(* IEC 61131-3 sources: CodesysTest/alpha/export/FBs/Components/Motors/Applied Motion/FB_AppliedMotionBagDeliveryMotor_1.pou, 13 files *)

(* ---- FB_AppliedMotionBagDeliveryMotor_1.pou.st ---- *)
(*#-#-#-#-#-#-#-#-#-#---Declaration---#-#-#-#-#-#-#-#-#-#-#-#-#*)

FUNCTION_BLOCK FB_AppliedMotionBagDeliveryMotor_1 EXTENDS FB_AppliedMotionStepServoEIPBase
VAR_INPUT
	ack : BOOL;
	placement : BAG_DELIVERY_MOTOR_PLACEMENT;
	intercommunications : BAG_DELIVERY_MOTOR_INTERCOMMUNICATION;
END_VAR
VAR_OUTPUT
	ackRequest : BOOL;
	tensionFault : BOOL;
END_VAR
VAR
	_moveDistance : BOOL;
	_moveFinal : BOOL;
	_moveDone : BOOL;
	_delayTimer : TON := (PT := T#10MS);
	_moveDistanceState : AMP_EIP_MOVE_INITIAL_STATES;
	_moveDistanceFinalState : AMP_EIP_MOVE_INITIAL_STATES;
	_tensionFaultDwellTimer : TON;
END_VAR
(*#-#-#-#-#-#-#-#-#-#---Implementation---#-#-#-#-#-#-#-#-#-#-#-#-#*)

(* ---- Execute.m.st ---- *)
(*#-#-#-#-#-#-#-#-#-#---Declaration---#-#-#-#-#-#-#-#-#-#-#-#-#*)

METHOD Execute
VAR_INPUT
END_VAR

(*#-#-#-#-#-#-#-#-#-#---Implementation---#-#-#-#-#-#-#-#-#-#-#-#-#*)

//
SUPER^.Execute();

// Used in state engine to delay between moves
_delayTimer();

// If motor velocity is greater then threshold for 2 seconds, fault
_tensionFaultDwellTimer(IN := ABS(velocity) > VELOCITY_THRESHOLD_FOR_TENSION_FAULT);
IF _tensionFaultDwellTimer.Q AND NOT HMIData.enableDryCycle THEN
	tensionFault := TRUE;
END_IF

// Clear Params
IF _restoreToDefault THEN
	_restoreToDefault := FALSE;
	_state := BAG_DELIVERY_MOVE_STATES.Idle;
	commandSuccessful := FALSE;
	tensionFault := FALSE;
	ackRequest := FALSE;
	ack := FALSE;
END_IF

//
CASE _state OF
	BAG_DELIVERY_MOVE_STATES.Idle:
		IF _moveDistance THEN
			_moveDistance := FALSE;
			_state := BAG_DELIVERY_MOVE_STATES.SetToPointToPointMode;
			commandSuccessful := FALSE;
		END_IF

	BAG_DELIVERY_MOVE_STATES.SetToPointToPointMode:
		IF EIP THEN
			IF RearMotor THEN
				TriggerPointToPointMode();
			END_IF
			IF commandSuccessful OR NOT RearMotor THEN
				commandSuccessful := FALSE;
				_state := BAG_DELIVERY_MOVE_STATES.AckPointToPointMode;
			END_IF
		ELSIF NOT EIP THEN
			sclCommand := SCL_SO;
			parameter1 := O2_H;
			commands.SendHostCommand := TRUE;
			IF commandSuccessful THEN
				commandSuccessful := FALSE;
				_state := BAG_DELIVERY_MOVE_STATES.WaitAfterMovingMotor;
			END_IF
		END_IF

	BAG_DELIVERY_MOVE_STATES.WaitAfterSettingOutputOff:
		IF commandSuccessful THEN
			_state := BAG_DELIVERY_MOVE_STATES.MoveMotor;
		END_IF

	BAG_DELIVERY_MOVE_STATES.AckPointToPointMode:
		_delayTimer.PT := T#10MS;
		_delayTimer.IN := TRUE;
		IF _delayTimer.Q THEN
			ackRequest := TRUE; // Request acknowledgment from parent class
			IF ack THEN // Parent class acknowledges this motor and sibling are ready to move
				ackRequest := FALSE;
				_delayTimer.IN := FALSE;
				_state := BAG_DELIVERY_MOVE_STATES.MoveMotor;
			END_IF
		END_IF

	BAG_DELIVERY_MOVE_STATES.MoveMotor:
		FeedToLength();
		_state := BAG_DELIVERY_MOVE_STATES.WaitAfterMovingMotor;

	BAG_DELIVERY_MOVE_STATES.WaitAfterMovingMotor:
		IF NOT _moveFinal THEN
			IF commandSuccessful THEN
				commandSuccessful := FALSE;
				_moveDone := TRUE;
				_state := BAG_DELIVERY_MOVE_STATES.Idle;
			END_IF
		ELSE
			IF commandSuccessful AND InPosition THEN
				_delayTimer.PT := T#10MS;
				_delayTimer.IN := TRUE;
				IF _delayTimer.Q THEN
					_delayTimer.IN := FALSE;
					commandSuccessful := FALSE;
					_state := BAG_DELIVERY_MOVE_STATES.SetToTorqueMode;
				END_IF
			END_IF
		END_IF

	BAG_DELIVERY_MOVE_STATES.SetToTorqueMode:
		IF EIP THEN
			IF RearMotor THEN
				TriggerTorqueMode();
			END_IF
			IF commandSuccessful OR NOT RearMotor THEN
				commandSuccessful := FALSE;
				_state := BAG_DELIVERY_MOVE_STATES.WaitAfterSettingOutputOn;
			END_IF
		ELSE
			TriggerTorqueMode();
			_state := BAG_DELIVERY_MOVE_STATES.WaitAfterSettingOutputOn;
		END_IF

	BAG_DELIVERY_MOVE_STATES.WaitAfterSettingOutputOn:
		IF EIP THEN
			_delayTimer.PT := T#10MS;
			_delayTimer.IN := TRUE;
			IF _delayTimer.Q THEN
				_moveDone := TRUE;
				_moveFinal := FALSE;
				_delayTimer.IN := FALSE;
				_state := BAG_DELIVERY_MOVE_STATES.Idle;
			END_IF
		ELSE
			IF commandSuccessful THEN
				_moveDone := TRUE;
				_state := BAG_DELIVERY_MOVE_STATES.Idle;
				commandSuccessful := FALSE;
			END_IF
		END_IF
END_CASE

(* ---- FeedToLength.m.st ---- *)
(*#-#-#-#-#-#-#-#-#-#---Declaration---#-#-#-#-#-#-#-#-#-#-#-#-#*)

METHOD FeedToLength
VAR_INPUT
END_VAR
(*#-#-#-#-#-#-#-#-#-#---Implementation---#-#-#-#-#-#-#-#-#-#-#-#-#*)

//
sclCommand := 16#0;
parameter1 := 16#0;
commandSuccessful := FALSE;
commands.FeedToLength := TRUE;

(* ---- Initialize.m.st ---- *)
(*#-#-#-#-#-#-#-#-#-#---Declaration---#-#-#-#-#-#-#-#-#-#-#-#-#*)

METHOD Initialize
VAR_INPUT
END_VAR
(*#-#-#-#-#-#-#-#-#-#---Implementation---#-#-#-#-#-#-#-#-#-#-#-#-#*)

//
_initialize := TRUE;

(* ---- MoveDistance.m.st ---- *)
(*#-#-#-#-#-#-#-#-#-#---Declaration---#-#-#-#-#-#-#-#-#-#-#-#-#*)

METHOD MoveDistance
VAR_INPUT
    distance : REAL;    // Distance to move in inches
    acceleration : INT; // Acceleration in RPM/sec
    deceleration : INT; // Deceleration in RPM/sec
    velocity : INT;     // Velocity in .25RPM
END_VAR(*#-#-#-#-#-#-#-#-#-#---Implementation---#-#-#-#-#-#-#-#-#-#-#-#-#*)

//
IF _initialize OR placement = BAG_DELIVERY_MOTOR_PLACEMENT.Rear AND interconnect = BAG_DELIVERY_IC.CBL THEN
	RETURN;
END_IF

//
_moveDone := FALSE;
_moveDistance := TRUE;
_state := BAG_DELIVERY_MOVE_STATES.Idle;

//
distanceToMoveInSteps := REAL_TO_DINT((distance) * stepsPerInchSetpoint);
IF reversePolarity THEN
    distanceToMoveInSteps := distanceToMoveInSteps * -1;
END_IF

//
commandSuccessful := FALSE;
pointToPointAccelSetpoint := acceleration;
pointToPointDecelSetpoint := deceleration;
currentLimit := defaultCurrentSetpoint;
velocitySetpoint := velocity;

(* ---- MoveDistanceFinal.m.st ---- *)
(*#-#-#-#-#-#-#-#-#-#---Declaration---#-#-#-#-#-#-#-#-#-#-#-#-#*)

METHOD MoveDistanceFinal
VAR_INPUT
    distance : REAL;        //Distance to move in inches
    acceleration : INT;        //Acceleration in RPM/sec
    deceleration : INT;        //Deceleration in RPM/sec
    velocity : INT;            //Velocity in .25RPM
END_VAR

VAR
	_movefin: BOOL;
END_VAR(*#-#-#-#-#-#-#-#-#-#---Implementation---#-#-#-#-#-#-#-#-#-#-#-#-#*)

//
_moveDone := FALSE;
_moveFinal := TRUE;
_stateFinal := BAG_DELIVERY_MOVE_STATES.Idle;

//
distanceToMoveInSteps := REAL_TO_DINT((distance) * stepsPerInchSetpoint);
IF reversePolarity THEN
    distanceToMoveInSteps := distanceToMoveInSteps * -1;
END_IF

//
commandSuccessful := FALSE;
pointToPointAccelSetpoint := acceleration;
pointToPointDecelSetpoint := deceleration;
currentLimit := defaultCurrentSetpoint;
velocitySetpoint := velocity;

(* ---- PrepareForCommand.m.st ---- *)
(*#-#-#-#-#-#-#-#-#-#---Declaration---#-#-#-#-#-#-#-#-#-#-#-#-#*)

METHOD PrepareForCommand
VAR_INPUT
END_VAR
(*#-#-#-#-#-#-#-#-#-#---Implementation---#-#-#-#-#-#-#-#-#-#-#-#-#*)

commandSuccessful := FALSE;

(* ---- SetRearMotorToPoint2Point.m.st ---- *)
(*#-#-#-#-#-#-#-#-#-#---Declaration---#-#-#-#-#-#-#-#-#-#-#-#-#*)

METHOD SetRearMotorToPoint2Point
VAR_INPUT
END_VAR
(*#-#-#-#-#-#-#-#-#-#---Implementation---#-#-#-#-#-#-#-#-#-#-#-#-#*)

commandSuccessful := FALSE;
ExecuteStoredProgram(2);

(* ---- SetRearMotorTorqueValue.m.st ---- *)
(*#-#-#-#-#-#-#-#-#-#---Declaration---#-#-#-#-#-#-#-#-#-#-#-#-#*)

METHOD SetRearMotorTorqueValue
VAR_INPUT
	torque : DINT;
END_VAR
(*#-#-#-#-#-#-#-#-#-#---Implementation---#-#-#-#-#-#-#-#-#-#-#-#-#*)

sclCommand := 16#4743; // GC (Current Command)
parameter1 := torque;

commandSuccessful := FALSE;
commands.SendHostCommand := TRUE;

(* ---- SetRearMotorToTorqueMode.m.st ---- *)
(*#-#-#-#-#-#-#-#-#-#---Declaration---#-#-#-#-#-#-#-#-#-#-#-#-#*)

METHOD SetRearMotorToTorqueMode
VAR_INPUT
END_VAR
(*#-#-#-#-#-#-#-#-#-#---Implementation---#-#-#-#-#-#-#-#-#-#-#-#-#*)

commandSuccessful := FALSE;
ExecuteStoredProgram(3);

(* ---- SetTorqueValue.m.st ---- *)
(*#-#-#-#-#-#-#-#-#-#---Declaration---#-#-#-#-#-#-#-#-#-#-#-#-#*)

METHOD SetTorqueValue
VAR_INPUT
	torque : DINT;
END_VAR
(*#-#-#-#-#-#-#-#-#-#---Implementation---#-#-#-#-#-#-#-#-#-#-#-#-#*)

sclCommand := 16#4743; // GC (Current Command)
parameter1 := torque;

commandSuccessful := FALSE;
commands.SendHostCommand := TRUE;

(* ---- TriggerPointToPointMode.m.st ---- *)
(*#-#-#-#-#-#-#-#-#-#---Declaration---#-#-#-#-#-#-#-#-#-#-#-#-#*)

METHOD TriggerPointToPointMode
VAR_INPUT
END_VAR

(*#-#-#-#-#-#-#-#-#-#---Implementation---#-#-#-#-#-#-#-#-#-#-#-#-#*)

parameter1 := POINT2POINT_MODE_PARAM_ID;
commands.SendQAndExecute := TRUE;

(* ---- TriggerTorqueMode.m.st ---- *)
(*#-#-#-#-#-#-#-#-#-#---Declaration---#-#-#-#-#-#-#-#-#-#-#-#-#*)

METHOD TriggerTorqueMode
VAR_INPUT
END_VAR
VAR CONSTANT
	TORQUE_MODE_ID : INT := 2;
END_VAR
(*#-#-#-#-#-#-#-#-#-#---Implementation---#-#-#-#-#-#-#-#-#-#-#-#-#*)

parameter1 := TORQUE_MODE_ID;
commands.SendQAndExecute := TRUE;
